PROGRAM D_1_CSV
VAR
	
	fbWriteEventsHistoryToCSV			: FB_WriteDataToCSV;

	DATECHANGETEST		: STRING;
	btest				: ARRAY[0..10] OF BOOL;
	i					: DINT;
	rPulsTrigger		: R_TRIG;
	fPulsTrigger		: F_TRIG;
	Counter				: CTU;

END_VAR

stCSV_EventsHistory.aDataLength					:= 200;

IF stCSV_EventsHistory.nDataHistoryIndex = 0 THEN
	
	stCSV_EventsHistory.bAcknowledge  			:= TRUE;
	
ELSE stCSV_EventsHistory.bAcknowledge  			:= FALSE;

END_IF

fbWriteEventsHistoryToCSV(

					//INPUTS
					bWriteData 					:= stCSV_EventsHistory.bWriteData,
					sFileNamePath				:= 'C:\Users\Sebastian.Ulloa\Desktop\CSV_TEST\newtest\',
					aData						:=	astEventsHistory,
					aDataLength 				:=	stCSV_EventsHistory.aDataLength,
					sDate						:= DATECHANGETEST,//sSystemDate,
					nMAX_CSV_ROWS				:=1000,
					nMAX_CSV_COLUMNS			:= 4,
					bAcknowledge				:= stCSV_EventsHistory.bAcknowledge,
					
					//OUTPUTS
					bBusy						=> stCSV_EventsHistory.bBusy,
					bError						=> stCSV_EventsHistory.bError,
					bDataWrited					=> stCSV_EventsHistory.bDataWrited
					
						
);

rPulsTrigger( CLK := stPuls.bFlash10Hz);


Counter(CU := stPuls.bFlash10Hz, RESET := Counter.CV > 3,);
IF btest[0] THEN
IF Counter.CV = 0 THEN
		
		bResetTest							:= FALSE;

		bTestFlag[0]						:= TRUE;
		
ELSIF Counter.CV = 1 THEN
		
		bTestFlag[1]						:= TRUE;
		
ELSIF Counter.CV = 2 THEN
		
		bTestFlag[2]						:= TRUE;
		
ELSIF Counter.CV = 3 THEN
	
		bTestFlag[0]						:= FALSE;
		bTestFlag[1]						:= FALSE;
		bTestFlag[2]						:= FALSE;
		bResetTest							:= TRUE;
		
END_IF
END_IF

END_PROGRAM

(* stored: Version 1.1.0.1, ProductVersion 3.1.4024.13
   POU D_1_CSV: Id {c1a3edab-978c-4461-bdb4-a2aa1b50049c}, SpecialFunc None *)
